INTERFACE I_Ipro_MotorPower

PROPERTY Active : bool
GET
END_GET
END_PROPERTY

PROPERTY Busy : bool
GET
END_GET
END_PROPERTY

PROPERTY ControlMode : E_IProCtrlMode
GET
END_GET
SET
END_SET
END_PROPERTY

PROPERTY ControlModeSwitchCmd : bool
GET
END_GET
END_PROPERTY

PROPERTY CurrentMode : E_IProCurrentMode
GET
END_GET
END_PROPERTY

PROPERTY Enable : bool
GET
END_GET
END_PROPERTY

PROPERTY Error : Reference to Bool
GET
END_GET
END_PROPERTY

PROPERTY ErrorID : REFERENCE TO INT
GET
END_GET
END_PROPERTY

PROPERTY InPosition : bool
GET
END_GET
END_PROPERTY

PROPERTY IsInTorque : bool
GET
END_GET
END_PROPERTY

PROPERTY isStop : bool
GET
END_GET
END_PROPERTY

PROPERTY MaxSpeed : lreal// large than 0
GET
END_GET
SET
END_SET
END_PROPERTY

PROPERTY MaxTorque : Lreal// // % larger than 0
GET
END_GET
SET
END_SET
END_PROPERTY

METHOD MR_Abort : BOOL
END_METHOD

METHOD MR_Home : BOOL // control mode must have Position Mode // actually it the same as MOVE absolute 
VAR_INPUT
	lrHomePosition : LREAL;
END_VAR
END_METHOD

(*this must be called 2 times, first: after set All parram in "SetBefor Init" folder and before run FBModbusMaster
							 second : after Modbusmster running and state machine in Init state.*)
METHOD MR_Init : BOOL// need to set control mode carefully, the control mode only work correct if you set p0.03 and restart the driver, and there for if you change control mode cmd during driver power ON, the control mode will not effect
END_METHOD

METHOD MR_MoveAbsolute : BOOL // control mode must have Position Mode
VAR_INPUT
	lrAbsolutePosition : LREAL;
END_VAR
END_METHOD

METHOD MR_MoveTorque : BOOL // control mode must have torque Mode
VAR_INPUT
	lrTorque	: LREAL;// must smaller than max torque
END_VAR
END_METHOD

METHOD MR_Reset : BOOL// can't not use this method because i didn't find way to reset
END_METHOD

METHOD MR_Stop : BOOL
END_METHOD

PROPERTY NagativePositionLimit : lreal
GET
END_GET
SET
END_SET
END_PROPERTY

PROPERTY PositionCmd : lreal
GET
END_GET
END_PROPERTY

PROPERTY PositionFeedBack : lreal
GET
END_GET
END_PROPERTY

PROPERTY PositionPositiveLimit : lreal
GET
END_GET
SET
END_SET
END_PROPERTY

PROPERTY SpeedCmd : LREAL // r/ minute
GET
END_GET
SET
END_SET
END_PROPERTY

PROPERTY SpeedFeedback : Lreal
GET
END_GET
END_PROPERTY

PROPERTY State : E_IPro_State
GET
END_GET
END_PROPERTY

PROPERTY Status : E_IProStatus
GET
END_GET
END_PROPERTY

PROPERTY TorqueCmd : lreal // %
GET
END_GET
END_PROPERTY

PROPERTY TorqueFeedback : lreal
GET
END_GET
END_PROPERTY

END_INTERFACE

(* stored: Version 1.1.0.1, ProductVersion 3.1.4024.12
   Itf I_Ipro_MotorPower: Id {c543df3e-e5ff-44c0-9d7a-938f099a67e7}
   Folder Parameters: Id {3d07359b-7e01-4eec-be43-8ab90aa28b60}
   Folder Requests: Id {c8788767-5005-4ab6-b433-64c9b2c00ae9}
   Folder SetBeforInit: Id {519a0f74-3e00-4d6f-af83-406953db9c88}
   Folder Status: Id {fe6257c1-1992-46da-9524-a9cc203bc5d5}
   Property Active: Id {f817ac78-9bed-4682-9538-a71cee528901}
   Get Get: Id {2a1910c4-ef7b-4639-9ffa-05ba33b47426}
   Property Busy: Id {50161faf-ccd5-432c-8d8e-54363d25b887}
   Get Get: Id {1ba27e72-5898-4d15-84f8-7c50a997053e}
   Property ControlMode: Id {5c12d86d-b455-4138-a387-4e3396dbda11}
   Get Get: Id {5b73fb7c-1902-427d-bf0d-f973df4d71ff}
   Set Set: Id {33b50898-7b34-4303-8ffb-dbbfaa9beb64}
   Property ControlModeSwitchCmd: Id {995b851c-f54b-452d-b650-96e6126d69ba}
   Get Get: Id {099810d6-30b7-406a-be97-7e8c21b028d3}
   Property CurrentMode: Id {d84910ca-4b79-4d9f-90c3-82428d7b6a84}
   Get Get: Id {aa13d564-0182-4695-8580-5d6c5ef5f081}
   Property Enable: Id {72b6a9dc-f1c0-4f36-a765-989f11faf8c4}
   Get Get: Id {e180f9e9-2500-4f07-a812-4390f2adc6dd}
   Property Error: Id {41a7854b-d106-4a4f-b550-956699843a93}
   Get Get: Id {cf5ebeb1-1f65-41c0-908b-aa65d1a49d3b}
   Property ErrorID: Id {eba52626-6e7b-4c80-b8cb-89fdc9cbc485}
   Get Get: Id {1ae1f15b-216f-4eaf-b327-5eb816d08fb7}
   Property InPosition: Id {5fe03aee-4d3a-46d4-8c8a-88f74409c2bb}
   Get Get: Id {e234b7ec-7441-4708-88d1-891507fcf1b8}
   Property IsInTorque: Id {69564cc0-27b1-42af-abb9-792845f9c43a}
   Get Get: Id {526056bc-4016-47ba-aea9-fc8ffd277812}
   Property isStop: Id {e5e4fc3e-44cf-4fb6-98e0-4dac1876084d}
   Get Get: Id {1ec42008-8ab0-4547-a1c1-7f10f9154584}
   Property MaxSpeed: Id {1c282d17-8ce7-43ae-944e-75f36051ea5c}
   Get Get: Id {31c81d87-89bc-4c62-9dad-4a0d54c7272e}
   Set Set: Id {f38813d8-4d61-4108-b987-18d3e027f8ba}
   Property MaxTorque: Id {7448fa9f-773b-46c8-ba83-8bd1634ebf62}
   Get Get: Id {aa4a9bd8-3afe-4dcc-84c4-d66be1481026}
   Set Set: Id {edf579d8-3c4a-4f80-ab04-9a879a1ec1c3}
   Method MR_Abort: Id {6b7355ea-a230-4fcd-b38c-196eca9c8280}
   Method MR_Home: Id {5e365130-9ee2-455f-8ef4-c19767f3ec36}
   Method MR_Init: Id {8da68057-161c-467e-bc76-2298ad85c346}
   Method MR_MoveAbsolute: Id {fc54e95e-5f3e-4c7c-ace7-df079eed0c41}
   Method MR_MoveTorque: Id {a9c8bc9a-6b60-4f2b-a03f-5dfe2cc21378}
   Method MR_Reset: Id {9b1e22f7-b5dd-44b1-99bd-8ba0419d70ad}
   Method MR_Stop: Id {8651239c-6ccc-4a36-bf17-5823b0334d66}
   Property NagativePositionLimit: Id {1176fd52-4e49-4c33-a209-df343cb6db4e}
   Get Get: Id {e022ae6b-4f6c-435d-b6ea-9f8ba7a85ffd}
   Set Set: Id {194e4f37-1796-46c7-8fda-2e3a37959acf}
   Property PositionCmd: Id {ecabd0b5-430e-4546-bc56-d9b8d7ae0a51}
   Get Get: Id {ec5ce21c-eb4e-45eb-9d2d-42b7d08941ae}
   Property PositionFeedBack: Id {1b7147fc-2525-485b-b645-4e4d3feb4a2c}
   Get Get: Id {9eadf0d0-692b-4972-a7ec-339b1a7afe05}
   Property PositionPositiveLimit: Id {65991d73-3f16-4967-8796-644e6cd77d11}
   Get Get: Id {0b43bb6f-86db-460e-8961-614feac12680}
   Set Set: Id {040a727d-4353-409a-8910-a8c310f40775}
   Property SpeedCmd: Id {80513a53-e5ac-4fb3-ad33-69f72acf349e}
   Get Get: Id {fa8b144c-319b-4d92-acd4-51e9b0327678}
   Set Set: Id {810f51ce-a8a0-416b-bda2-874d895a9a3b}
   Property SpeedFeedback: Id {7a656d80-a974-494a-9e99-bd618898dff7}
   Get Get: Id {354d87af-3697-433b-9dba-7399108512b9}
   Property State: Id {f7ee26ed-5e4d-4e8f-bf4c-d3955bafcb44}
   Get Get: Id {d84e70ef-3968-4a2d-aaa6-eb84051d49f4}
   Property Status: Id {3b352231-6273-494b-ae1d-fdd8f800a88c}
   Get Get: Id {12247c6d-0791-4708-8e5f-74b6fe498162}
   Property TorqueCmd: Id {510b39de-1542-4b73-98d5-a4802991c79b}
   Get Get: Id {c96c232a-497b-49ac-ad09-bca288efa079}
   Property TorqueFeedback: Id {27846add-514c-49a9-82e0-2d58e0d26b6a}
   Get Get: Id {369e6f3f-0f94-431c-bc3e-be5a53313627} *)
